(* IEC 61131-3 sources: AXOpen/src/core/app/src/Examples/AXOpen.AxoMomentaryTask, 2 files *)

(* ---- AxoMomentaryTaskDocuExample.st ---- *)
USING AXOpen.Core;

NAMESPACE AxoMomentaryTaskExamples
    {S7.extern=ReadWrite}
    CLASS AxoMomentaryTaskDocuExample EXTENDS  AXOpen.Core.AxoContext
        VAR PUBLIC
            {#ix-set:AttributeName = "<#Momentary task example#>"}
            {#ix-set:AttributeStateOnDesc = "<#Currently On#>"}
            {#ix-set:AttributeStateOffDesc = "<#Currently Off#>"}
            _myMomentaryTask : AxoMomentaryTask;
        END_VAR

        METHOD PUBLIC Initialize
            // Initialization of the context needs to be called first
            // It does not need to be called cyclically, just once
            THIS.InitializeRootObject(_myMomentaryTask);
        END_METHOD

        METHOD PROTECTED OVERRIDE Main
            // Cyclicall call of the Run method
            THIS.InitializeRootObject(_myMomentaryTask);
            _myMomentaryTask.Run();
        END_METHOD

        METHOD Examples

        //<AxoMomentaryTaskIsSwitchedOn>
        IF _myMomentaryTask.IsSwitchedOn() THEN
            ; // do something
        END_IF;
        //</AxoMomentaryTaskIsSwitchedOn>

        //<AxoMomentaryTaskIsSwitchedOff>
        IF _myMomentaryTask.IsSwitchedOff() THEN
            ; // do something
        END_IF;
        //</AxoMomentaryTaskIsSwitchedOff>
        END_METHOD
    END_CLASS

    //<AxoMomentaryTaskEventLikeMethods>
    {S7.extern=ReadWrite}
    CLASS MyMomentaryTaskExample Extends AxoMomentaryTask
        VAR
            OnSwitchedOnCounter : ULINT;
            OnSwitchedOffCounter : ULINT;
            OnStateChangedCounter : ULINT;
            SwitchOnExecutionCounter : ULINT;
            SwitchOffExecutionCounter : ULINT;
        END_VAR

        METHOD PROTECTED OVERRIDE OnSwitchedOn
            OnSwitchedOnCounter := OnSwitchedOnCounter + ULINT#1;
        END_METHOD

        METHOD PROTECTED OVERRIDE OnSwitchedOff
            OnSwitchedOffCounter := OnSwitchedOffCounter + ULINT#1;
        END_METHOD

        METHOD PROTECTED OVERRIDE OnStateChanged
            OnStateChangedCounter := OnStateChangedCounter + ULINT#1;
        END_METHOD

        METHOD PROTECTED OVERRIDE SwitchedOn
            SwitchOnExecutionCounter := SwitchOnExecutionCounter + ULINT#1;
        END_METHOD

        METHOD PROTECTED OVERRIDE SwitchedOff
            SwitchOffExecutionCounter := SwitchOffExecutionCounter + ULINT#1;
        END_METHOD
    END_CLASS
    //</AxoMomentaryTaskEventLikeMethods>
END_NAMESPACE

(* ---- AxoMomentaryTaskExample.st ---- *)
USING AXOpen.Core;

NAMESPACE AxoMomentaryTaskExamples

    {S7.extern=ReadWrite}
    CLASS PUBLIC AxoMomentaryTaskExample EXTENDS AXOpen.Core.AxoMomentaryTask
        VAR PUBLIC
            {#ix-set: AttributeName = "<#Disable#>"}
            Disable : BOOL;
            {#ix-set:AttributeName = "<#OnSwitchedOn counter#>"}
            OnSwitchedOnCounter : ULINT;
            {#ix-set:AttributeName = "<#OnSwitchedOff counter#>"}
            OnSwitchedOffCounter : ULINT;
            {#ix-set:AttributeName = "<#OnStateChanged counter#>"}
            OnStateChangedCounter : ULINT;
            {#ix-set:AttributeName = "<#While SwitchedOn counter#>"}
            SwitchOnExecutionCounter : ULINT;
            {#ix-set:AttributeName = "<#While SwitchedOff counter#>"}
            SwitchOffExecutionCounter : ULINT;
        END_VAR

        METHOD PROTECTED OVERRIDE OnSwitchedOn
            OnSwitchedOnCounter := OnSwitchedOnCounter + ULINT#1;
        END_METHOD

        METHOD PROTECTED OVERRIDE OnSwitchedOff
            OnSwitchedOffCounter := OnSwitchedOffCounter + ULINT#1;
        END_METHOD

        METHOD PROTECTED OVERRIDE OnStateChanged
            OnStateChangedCounter := OnStateChangedCounter + ULINT#1;
        END_METHOD

        METHOD PROTECTED OVERRIDE SwitchedOn
            SwitchOnExecutionCounter := SwitchOnExecutionCounter + ULINT#1;
        END_METHOD

        METHOD PROTECTED OVERRIDE SwitchedOff
            SwitchOffExecutionCounter := SwitchOffExecutionCounter + ULINT#1;
        END_METHOD
    END_CLASS

    {S7.extern=ReadWrite}
    CLASS Tasks EXTENDS AXOpen.Core.AxoContext
        VAR PUBLIC
            {#ix-set:AttributeName = "Momentary task example"}
            MomentaryTaskExample :AxoMomentaryTaskExample;
       END_VAR

        METHOD PROTECTED OVERRIDE Main
            MomentaryTaskExample.InitializeWithContext(THIS);
            MomentaryTaskExample.SetIsDisabled(MomentaryTaskExample.Disable);
            MomentaryTaskExample.Run();

        END_METHOD
    END_CLASS
END_NAMESPACE
